FUNCTION_BLOCK FB_Conveyor IMPLEMENTS I_Conveyor
VAR_INPUT
END_VAR
VAR_OUTPUT
END_VAR
VAR
	//fbInverter		: FB_Inverter;
	bRunConveyor AT %Q* : BOOL;
	bIsRun		 AT %I* : BOOL;
END_VAR

PROPERTY IsRun : BOOL
GET
IsRun := bIsRun;
END_GET
END_PROPERTY

METHOD Start : BOOL
VAR_INPUT
END_VAR
bRunConveyor := TRUE;
END_METHOD

METHOD Stop : BOOL
VAR_INPUT
END_VAR
bRunConveyor := FALSE;
END_METHOD

END_FUNCTION_BLOCK

(* stored: Version 1.1.0.1, ProductVersion 3.1.4024.12
   POU FB_Conveyor: Id {fdb31384-3855-49d6-a7fb-6f97a622bab9}, SpecialFunc None
   Property IsRun: Id {3c39b5ee-9694-4031-a99a-23bb4f62aba8}
   Get Get: Id {7cff29e8-086b-4cbe-8df2-f839d46695d9}
   Method Start: Id {fd9da3d7-de72-4590-949e-5f2c0fb16ef4}
   Method Stop: Id {72ef631a-e78e-424b-a463-0de6b401e5f4} *)
